TYPE RX_Step_PC :
STRUCT
	Comandi      : WORD;		// Word (16 bit) ==> comandi (16 byte)
	ps		     : UINT;		// Nodo da raggiungere nello step
	dist	     : UINT;		// Distanza del Nodo da raggiungere (in cm)
	rall	     : UINT;		// Rallentamento specifico nello Step
	CmFree1		 : UINT;		
	CmFree2		 : UINT;		
	CmFree3		 : UINT;		
END_STRUCT
END_TYPE

(* stored: Version 1.1.0.1, ProductVersion 3.1.4024.11
   DUT RX_Step_PC: Id {27b611a3-9463-49a1-a94e-d3093b88337d} *)
